Staubli VAL3: robotStatusInq.pjx

Parameters version=s7.9.1 stackSize=5000 millimeterUnit=true
Program file=robotStatusInq.pgx
Program file=start.pgx
Program file=stop.pgx
Data file=robotStatusInq.dtx
Type name=RobotCfgStatus path=Disk://RobotController_Libs/RobotCfgStatus/RobotCfgStatus.pjx
Type name=RobotStatus path=Disk://RobotController_Libs/RobotStatus/RobotStatus.pjx
